Staubli VAL3: clkValve6.pgx

program clkValve6()
begin
  call toggleValve(6)
end
